// TIA Portal V21 export
DATA_BLOCK "HMI_DB"   // DB700
{ S7_Optimized_Access := 'TRUE' }
// stored: AutoNumber false, DBAccessibleFromWebserver false, MemoryReserve 100
   VAR
      MachineState { ExternalWritable := 'False'} : USInt;
      Device { ExternalAccessible := 'False'; ExternalVisible := 'False'; ExternalWritable := 'False'} : Struct
         Pump : Array[1..2] of "UDT_Device";
      END_STRUCT;
      Devices_Status { ExternalWritable := 'False'} : Struct
         Pump : Array[1..2] of Int;
      END_STRUCT;
   END_VAR
BEGIN
END_DATA_BLOCK
